(* PLC project marvel_guiding, Institute of Astronomy Onto 0.0.1 *)
(* stored: creationDateTime 2025-01-01T00:00:00.0, modificationDateTime 2025-01-01T00:00:00.0 *)

{attribute 'qualified_only'}
TYPE GuidingStates : (IDLE := 0, ACQUISITION := 1, GUIDING := 2);
END_TYPE

{attribute 'qualified_only'}
TYPE GuidingCameraParamSets : (INIT := 0, CONTINUOUS_IMAGING := 1, TRIGGER_IMAGING := 2);
END_TYPE

TYPE GuidingParts : STRUCT
  {attribute 'TcHmiSymbol.Show'}
  camera : GigECamera;
END_STRUCT;
END_TYPE

TYPE GuidingProcesses : STRUCT
  {attribute 'TcHmiSymbol.Show'}
  initialize : Process;  (* Start initializing *)
  {attribute 'TcHmiSymbol.Show'}
  reset : Process;  (* Reset any errors *)
  {attribute 'TcHmiSymbol.Show'}
  acquireTarget : GuidingAcquireTargetProcess;  (* Acquire the target *)
  {attribute 'TcHmiSymbol.Show'}
  startGuiding : GuidingStartGuidingProcess;  (* Start guiding *)
  {attribute 'TcHmiSymbol.Show'}
  stop : Process;  (* Stop guiding and acquisition *)
  {attribute 'TcHmiSymbol.Show'}
  setCameraParamSet : GuidingCameraParamSetProcess;  (* Set a parameter set *)
END_STRUCT;
END_TYPE

TYPE GuidingStatuses : STRUCT
  {attribute 'OPC.UA.DA' := '1'}
  {attribute 'OPC.UA.DA.Access' := '1'}
  {attribute 'TcHmiSymbol.Show'}
  init : InitializationStatus;
  {attribute 'OPC.UA.DA' := '1'}
  {attribute 'OPC.UA.DA.Access' := '1'}
  {attribute 'TcHmiSymbol.Show'}
  health : HealthStatus;
  {attribute 'OPC.UA.DA' := '1'}
  {attribute 'OPC.UA.DA.Access' := '1'}
  {attribute 'TcHmiSymbol.Show'}
  busy : BusyStatus;
END_STRUCT;
END_TYPE

TYPE GuidingConfig : STRUCT
  {attribute 'TcHmiSymbol.Show'}
  initExposureTime : LREAL;  (* Initial exposure time (in seconds) *)
  {attribute 'TcHmiSymbol.Show'}
  initAcquisitionFrameRate : LREAL;  (* Initial acquisition frame rate *)
  {attribute 'TcHmiSymbol.Show'}
  initGainDigital : LREAL;  (* Initial digital gain *)
  {attribute 'TcHmiSymbol.Show'}
  initGainAnalog : LREAL;  (* Initial analog gain *)
  {attribute 'TcHmiSymbol.Show'}
  initBinning : UDINT;  (* Initial analog gain *)
END_STRUCT;
END_TYPE

TYPE GuidingAcquireTargetProcessArgs : STRUCT
  {attribute 'TcHmiSymbol.Show'}
  vMag : LREAL;  (* Visual magnitude of target *)
END_STRUCT;
END_TYPE

TYPE GuidingStartGuidingProcessArgs : STRUCT
  {attribute 'TcHmiSymbol.Show'}
  vMag : LREAL;  (* Visual magnitude of target *)
END_STRUCT;
END_TYPE

TYPE GuidingCameraParamSetProcessArgs : STRUCT
  {attribute 'TcHmiSymbol.Show'}
  paramSet : GuidingCameraParamSets;  (* Parameter set *)
END_STRUCT;
END_TYPE

TYPE M_SM_Guiding : STRUCT
  {attribute 'TcHmiSymbol.Show'}
  actualStatus : STRING;
  {attribute 'TcHmiSymbol.Show'}
  centroidXAbsCoo : LREAL;
  {attribute 'TcHmiSymbol.Show'}
  centroidYAbsCoo : LREAL;
  {attribute 'TcHmiSymbol.Show'}
  centroidXRelCoo : LREAL;
  {attribute 'TcHmiSymbol.Show'}
  centroidYRelCoo : LREAL;
  {attribute 'TcHmiSymbol.Show'}
  stat : GuidingStatuses;
  {attribute 'TcHmiSymbol.Show'}
  parts : M_SM_GuidingParts;
  {attribute 'TcHmiSymbol.Show'}
  proc : M_SM_GuidingProcesses;
END_STRUCT;
END_TYPE

TYPE M_GuidingAcquireTargetProcess : STRUCT

END_STRUCT;
END_TYPE

TYPE M_GuidingStartGuidingProcess : STRUCT

END_STRUCT;
END_TYPE

TYPE M_GuidingCameraParamSetProcess : STRUCT

END_STRUCT;
END_TYPE

TYPE M_SM_GuidingParts : STRUCT
  {attribute 'TcHmiSymbol.Show'}
  camera : M_GigECamera;
END_STRUCT;
END_TYPE

TYPE M_SM_GuidingProcesses : STRUCT
  {attribute 'TcHmiSymbol.Show'}
  initialize : M_Process;
  {attribute 'TcHmiSymbol.Show'}
  reset : M_Process;
  {attribute 'TcHmiSymbol.Show'}
  acquireTarget : M_GuidingAcquireTargetProcess;
  {attribute 'TcHmiSymbol.Show'}
  startGuiding : M_GuidingStartGuidingProcess;
  {attribute 'TcHmiSymbol.Show'}
  stop : M_Process;
  {attribute 'TcHmiSymbol.Show'}
  setCameraParamSet : M_GuidingCameraParamSetProcess;
END_STRUCT;
END_TYPE

FUNCTION_BLOCK SM_Guiding
  VAR_OUTPUT
    {attribute 'OPC.UA.DA' := '1'}
    {attribute 'OPC.UA.DA.Access' := '1'}
    {attribute 'TcHmiSymbol.Show'}
    actualStatus : STRING;  (* Current status description *)
    {attribute 'TcHmiSymbol.Show'}
    {attribute 'OPC.UA.DA' := '1'}
    {attribute 'OPC.UA.DA.Access' := '1'}
    state : GuidingStates;  (* Actual guiding state *)
    {attribute 'TcHmiSymbol.Show'}
    {attribute 'OPC.UA.DA' := '1'}
    {attribute 'OPC.UA.DA.Access' := '1'}
    centroidXAbsCoo : LREAL;  (* Centroid X absolute coordinate *)
    {attribute 'TcHmiSymbol.Show'}
    {attribute 'OPC.UA.DA' := '1'}
    {attribute 'OPC.UA.DA.Access' := '1'}
    centroidYAbsCoo : LREAL;  (* Centroid Y absolute coordinate *)
    {attribute 'TcHmiSymbol.Show'}
    {attribute 'OPC.UA.DA' := '1'}
    {attribute 'OPC.UA.DA.Access' := '1'}
    centroidXRelCoo : LREAL;  (* Centroid X relative coordinate *)
    {attribute 'TcHmiSymbol.Show'}
    {attribute 'OPC.UA.DA' := '1'}
    {attribute 'OPC.UA.DA.Access' := '1'}
    centroidYRelCoo : LREAL;  (* Centroid Y relative coordinate *)
    {attribute 'TcHmiSymbol.Show'}
    stat : GuidingStatuses;  (* Statuses of the state machine *)
    {attribute 'TcHmiSymbol.Show'}
    parts : GuidingParts;  (* Parts of the state machine *)
    {attribute 'TcHmiSymbol.Show'}
    proc : GuidingProcesses;  (* Processes of the state machine *)
  END_VAR
  VAR_IN_OUT
    {attribute 'TcHmiSymbol.Show'}
    {attribute 'OPC.UA.DA' := '0'}
    {attribute 'TcHmiSymbol.Hide'}
    number : USINT;  (* Number of the unit (1-4) *)
    {attribute 'TcHmiSymbol.Show'}
    {attribute 'OPC.UA.DA' := '0'}
    {attribute 'TcHmiSymbol.Hide'}
    operator_ref : OperatorStatus;  (* Shared operator status *)
    {attribute 'TcHmiSymbol.Show'}
    {attribute 'OPC.UA.DA' := '0'}
    {attribute 'TcHmiSymbol.Hide'}
    activity_ref : ActivityStatus;  (* Shared activity status *)
    {attribute 'TcHmiSymbol.Show'}
    {attribute 'OPC.UA.DA' := '0'}
    {attribute 'TcHmiSymbol.Hide'}
    services_ref : Services;  (* Shared services *)
    {attribute 'TcHmiSymbol.Show'}
    {attribute 'OPC.UA.DA' := '0'}
    {attribute 'TcHmiSymbol.Hide'}
    config_ref : GuidingConfig;  (* Active configuration of the guiding *)
  END_VAR

            parts.camera();
stat.health := F_HealthStatus(
    superState := TRUE,
    isGood := parts.camera.stat.health = HealthStatus.good,
    hasWarning := parts.camera.stat.health = HealthStatus.warning);
stat.busy := F_BusyStatus(
    superState := TRUE,
    isBusy := parts.camera.stat.busy = BusyStatus.busy);
proc.initialize( isEnabled := (NOT(stat.init = InitializationStatus.locked)) AND ((stat.init = InitializationStatus.shutdown) OR ((stat.init = InitializationStatus.initializingFailed) OR (stat.init = InitializationStatus.initialized))) );
proc.reset( isEnabled := TRUE );
proc.acquireTarget( isEnabled := TRUE );
proc.startGuiding();
proc.stop( isEnabled := TRUE );
proc.setCameraParamSet( isEnabled := TRUE );

          
END_FUNCTION_BLOCK

FUNCTION_BLOCK GuidingAcquireTargetProcess EXTENDS BaseProcess
  VAR_INPUT
    {attribute 'OPC.UA.DA' := '1'}
    {attribute 'OPC.UA.DA.Access' := '3'}
    {attribute 'TcHmiSymbol.Show'}
    set : GuidingAcquireTargetProcessArgs;  (* Arguments to be set, before writing do_request TRUE *)
  END_VAR
  VAR_OUTPUT
    {attribute 'OPC.UA.DA' := '1'}
    {attribute 'OPC.UA.DA.Access' := '1'}
    {attribute 'TcHmiSymbol.Show'}
    get : GuidingAcquireTargetProcessArgs;  (* Arguments in use by the process, if do_request was accepted *)
  END_VAR

            IF do_request THEN
    do_request_result := request( vMag := set.vMag );
    do_request := FALSE;
END_IF;
SUPER^();

          

{attribute 'TcRpcEnable' := '1'}
METHOD start
  VAR_INPUT
    {attribute 'TcHmiSymbol.Show'}
    vMag : LREAL;  (* Visual magnitude of target *)
  END_VAR
                  THIS^.get.vMag := vMag;
THIS^.stat.busy := BusyStatus.busy;
THIS^.stat.health := HealthStatus.good;

                
END_METHOD

{attribute 'TcRpcEnable' := '1'}
METHOD request : RequestResults
  VAR_INPUT
    {attribute 'TcHmiSymbol.Show'}
    vMag : LREAL;  (* Visual magnitude of target *)
  END_VAR
                  IF THIS^.stat.enabled = EnabledStatus.enabled THEN
    request := RequestResults.ACCEPTED;
    THIS^.start( vMag := vMag );
ELSE
    request := RequestResults.REJECTED;
END_IF;

                
END_METHOD
END_FUNCTION_BLOCK

FUNCTION_BLOCK GuidingStartGuidingProcess EXTENDS BaseProcess
  VAR_INPUT
    {attribute 'OPC.UA.DA' := '1'}
    {attribute 'OPC.UA.DA.Access' := '3'}
    {attribute 'TcHmiSymbol.Show'}
    set : GuidingStartGuidingProcessArgs;  (* Arguments to be set, before writing do_request TRUE *)
  END_VAR
  VAR_OUTPUT
    {attribute 'OPC.UA.DA' := '1'}
    {attribute 'OPC.UA.DA.Access' := '1'}
    {attribute 'TcHmiSymbol.Show'}
    get : GuidingStartGuidingProcessArgs;  (* Arguments in use by the process, if do_request was accepted *)
  END_VAR

            IF do_request THEN
    do_request_result := request( vMag := set.vMag );
    do_request := FALSE;
END_IF;
SUPER^();

          

{attribute 'TcRpcEnable' := '1'}
METHOD start
  VAR_INPUT
    {attribute 'TcHmiSymbol.Show'}
    vMag : LREAL;  (* Visual magnitude of target *)
  END_VAR
                  THIS^.get.vMag := vMag;
THIS^.stat.busy := BusyStatus.busy;
THIS^.stat.health := HealthStatus.good;

                
END_METHOD

{attribute 'TcRpcEnable' := '1'}
METHOD request : RequestResults
  VAR_INPUT
    {attribute 'TcHmiSymbol.Show'}
    vMag : LREAL;  (* Visual magnitude of target *)
  END_VAR
                  IF THIS^.stat.enabled = EnabledStatus.enabled THEN
    request := RequestResults.ACCEPTED;
    THIS^.start( vMag := vMag );
ELSE
    request := RequestResults.REJECTED;
END_IF;

                
END_METHOD
END_FUNCTION_BLOCK

FUNCTION_BLOCK GuidingCameraParamSetProcess EXTENDS BaseProcess
  VAR_INPUT
    {attribute 'OPC.UA.DA' := '1'}
    {attribute 'OPC.UA.DA.Access' := '3'}
    {attribute 'TcHmiSymbol.Show'}
    set : GuidingCameraParamSetProcessArgs;  (* Arguments to be set, before writing do_request TRUE *)
  END_VAR
  VAR_OUTPUT
    {attribute 'OPC.UA.DA' := '1'}
    {attribute 'OPC.UA.DA.Access' := '1'}
    {attribute 'TcHmiSymbol.Show'}
    get : GuidingCameraParamSetProcessArgs;  (* Arguments in use by the process, if do_request was accepted *)
  END_VAR

            IF do_request THEN
    do_request_result := request( paramSet := set.paramSet );
    do_request := FALSE;
END_IF;
SUPER^();

          

{attribute 'TcRpcEnable' := '1'}
METHOD start
  VAR_INPUT
    {attribute 'TcHmiSymbol.Show'}
    paramSet : GuidingCameraParamSets;  (* Parameter set *)
  END_VAR
                  THIS^.get.paramSet := paramSet;
THIS^.stat.busy := BusyStatus.busy;
THIS^.stat.health := HealthStatus.good;

                
END_METHOD

{attribute 'TcRpcEnable' := '1'}
METHOD request : RequestResults
  VAR_INPUT
    {attribute 'TcHmiSymbol.Show'}
    paramSet : GuidingCameraParamSets;  (* Parameter set *)
  END_VAR
                  IF THIS^.stat.enabled = EnabledStatus.enabled THEN
    request := RequestResults.ACCEPTED;
    THIS^.start( paramSet := paramSet );
ELSE
    request := RequestResults.REJECTED;
END_IF;

                
END_METHOD
END_FUNCTION_BLOCK
